FUNCTION_BLOCK CTRL_SEMA (* Basic Function Block Type *)
  (* Standard: 61499-2 *)
  (* Version 0.3, 2009-09-15, JHC, Holobloc Inc, Changed transition priorities. *)
  (* Version 0.2, 2003-12-04, JHC, Rockwell Automation, Renamed for better indexing. *)
  (* Version 0.1, 2002-11-05, JHC, Rockwell Automation, Corrected missing ST element in Algorithm REQ. *)
  (* Version 0.0, 2000-05-30, JHC, Rockwell Automation *)
  PACKAGE fb.rt.DIAS;
  IMPORT fb.datatype.*;
  IMPORT fb.rt.*;
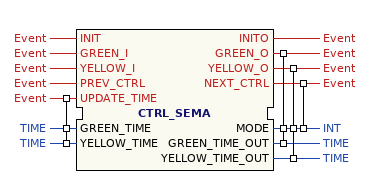
  EVENT_INPUT
    INIT; (* Initialization Request *)
    GREEN_I;
    YELLOW_I;
    PREV_CTRL;
    UPDATE_TIME WITH GREEN_TIME, YELLOW_TIME;
  END_EVENT
  EVENT_OUTPUT
    INITO; (* Initialization Confirm *)
    GREEN_O WITH MODE, GREEN_TIME_OUT;
    YELLOW_O WITH MODE, YELLOW_TIME_OUT;
    NEXT_CTRL WITH MODE;
  END_EVENT
  VAR_INPUT
    GREEN_TIME : TIME;
    YELLOW_TIME : TIME;
  END_VAR
  VAR_OUTPUT
    MODE : INT;
    GREEN_TIME_OUT : TIME;
    YELLOW_TIME_OUT : TIME;
  END_VAR
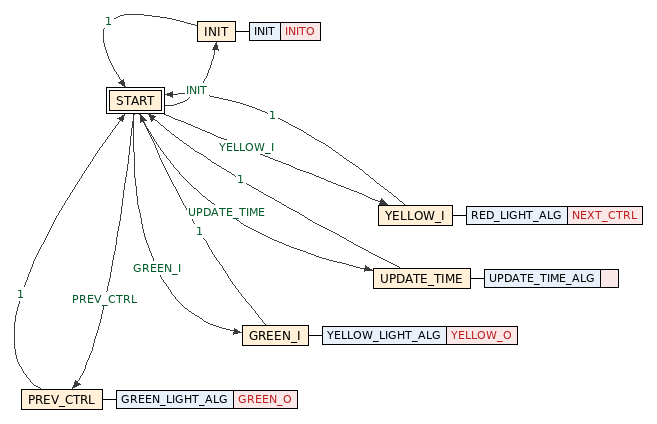
  EC_STATES
    START; (* Initial State *)
    INIT : INIT -> INITO; (* Initialization *)
    GREEN_I : YELLOW_LIGHT_ALG -> YELLOW_O;
    YELLOW_I : RED_LIGHT_ALG -> NEXT_CTRL;
    PREV_CTRL : GREEN_LIGHT_ALG -> GREEN_O;
    UPDATE_TIME : UPDATE_TIME_ALG;
  END_STATES
  EC_TRANSITIONS
    INIT TO START := 1;
    START TO INIT := INIT;
    START TO PREV_CTRL := PREV_CTRL;
    PREV_CTRL TO START := 1;
    START TO GREEN_I := GREEN_I;
    GREEN_I TO START := 1;
    START TO YELLOW_I := YELLOW_I;
    YELLOW_I TO START := 1;
    START TO UPDATE_TIME := UPDATE_TIME;
    UPDATE_TIME TO START := 1;
  END_TRANSITIONS
  ALGORITHM INIT IN ST: (* Initialization algorithm *)
MODE := 0;
  END_ALGORITHM
  ALGORITHM GREEN_LIGHT_ALG IN ST:
MODE := 2;
  END_ALGORITHM
  ALGORITHM YELLOW_LIGHT_ALG IN ST:
MODE := 1;
  END_ALGORITHM
  ALGORITHM RED_LIGHT_ALG IN ST:
MODE := 0;
  END_ALGORITHM
  ALGORITHM UPDATE_TIME_ALG IN ST:
GREEN_TIME_OUT := GREEN_TIME;
YELLOW_TIME_OUT := YELLOW_TIME;
  END_ALGORITHM
END_FUNCTION_BLOCK
